PROGRAM MAIN
VAR
END_VAR

/////////////////////////////////////////////////
///    Update motor data from feedback PDO
/////////////////////////////////////////////////
motor_settings.motor_interfaces[0]();
motor_settings.motor_interfaces[1]();
/////////////////////////////////////////////////
///           Motor Scheduler Loop
/////////////////////////////////////////////////
motor_settings.pp_scheduler[0]();
motor_settings.csp_scheduler[0]();
motor_settings.hm_scheduler[0]();
motor_settings.pp_scheduler[1]();
motor_settings.csp_scheduler[1]();
motor_settings.hm_scheduler[1]();
/////////////////////////////////////////////////
///           Update Robot Interface
/////////////////////////////////////////////////
robot_settings.robot_interface();
robot_settings.robot_pp_scheduler();
robot_settings.robot_hm_scheduler();
robot_settings.robot_traj_scheduler();

END_PROGRAM

(* stored: Version 1.1.0.1, ProductVersion 3.1.4024.12
   POU MAIN: Id {02236a42-b994-4274-a556-f8eb89138d77}, SpecialFunc None *)
